{attribute addProperty BoxType "KL9505-0010"}
{attribute addProperty Id "Diag_1Diag_619B670300"}
{attribute addProperty CRC "1874494086"}
{attribute addProperty SizeInBites "0"}
{attribute addProperty SizeInBytes "0"}
TYPE KL_6FBA8286 :
STRUCT
	{attribute addProperty Name "Diag_1"}
	Diag_1 : Diag_619B6703;
END_STRUCT
END_TYPE

(* stored: Version 1.2.0.0, ProductVersion 3.1.4024.9
   DUT KL_6FBA8286: Id {24eb4f65-3c83-440a-9926-ca9c4efbb761} *)
